Fanuc KAREL source: kt00006.KL

-- PROVISIONAL review KL for V770-1; original PC SHA256 78dc7e765bdfd1797bcfb5f0298df01e11d94d1e10d5635a776eb767d460efef
-- Incomplete behavior may be omitted. Consult companion uncertainty JSON. Do not deploy.
PROGRAM KT00006
%NOLOCKGROUP
VAR
  I1 : INTEGER
  OUT : REAL
-- UNRESOLVED_DECL Y2 type=002018
BEGIN
  -- UNRESOLVED_PC offsets 5-16; opcodes 2E,23
  -- UNRESOLVED_PC offsets 21-35; opcodes 2E,22,9D,33,B2
  -- UNRESOLVED_PC offsets 40-63; opcodes 21,22,9D,33,B1,52,64,23
  -- UNRESOLVED_PC offsets 68-72; opcodes 7F
END KT00006
